SYSTEM ModbusExmpl
  (* Version 1.0, 2026-07-14, alex *)
  APPLICATION testttApp
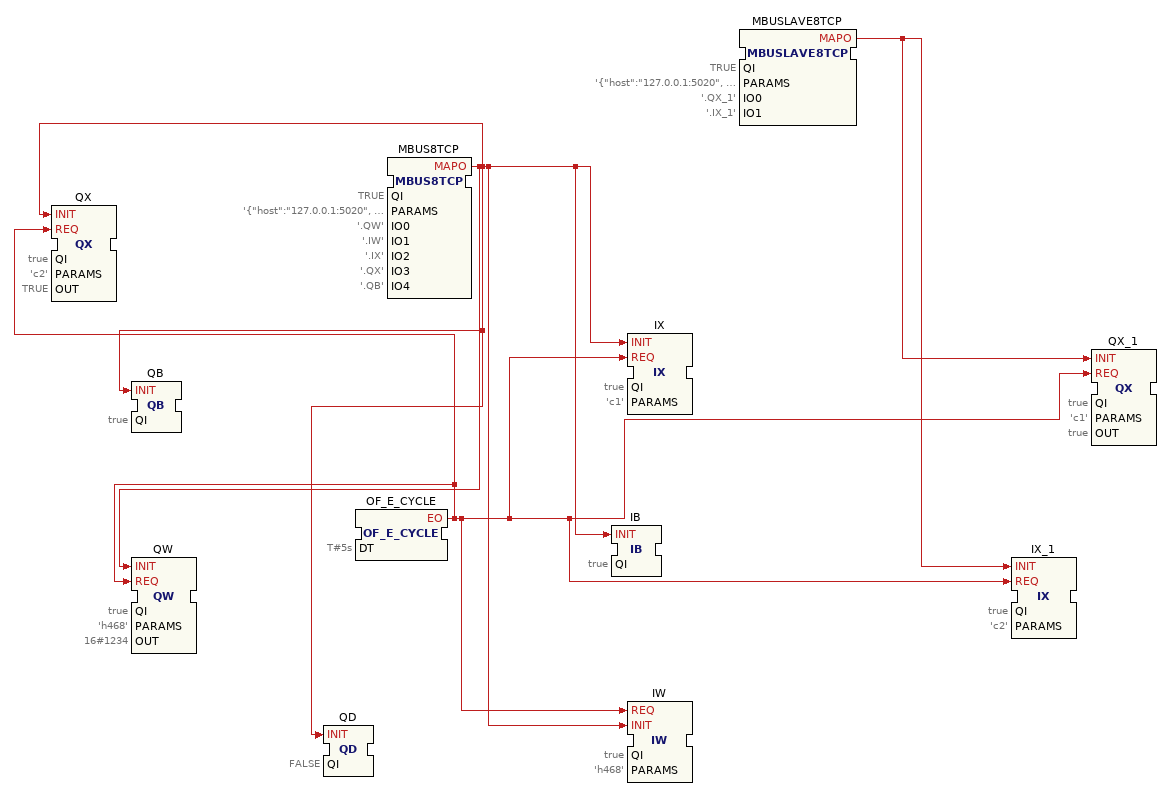
    FBS
      MBUS8TCP : MBUS8TCP(QI := TRUE, PARAMS := '{"host":"127.0.0.1:5020", "id":"1"}', IO0 := '.QW', IO1 := '.IW', IO2 := '.IX', IO3 := '.QX', IO4 := '.QB');
      MBUSLAVE8TCP : MBUSLAVE8TCP(QI := TRUE, PARAMS := '{"host":"127.0.0.1:5020", "id":"1"}', IO0 := '.QX_1', IO1 := '.IX_1');
      QX : QX(QI := true, PARAMS := 'c2', OUT := TRUE);
      QB : QB(QI := true);
      QD : QD(QI := FALSE);
      QW : QW(QI := true, PARAMS := 'h468', OUT := 16#1234);
      IX : IX(QI := true, PARAMS := 'c1');
      IB : IB(QI := true);
      IX_1 : IX(QI := true, PARAMS := 'c2');
      QX_1 : QX(QI := true, PARAMS := 'c1', OUT := true);
      OF_E_CYCLE : OF_E_CYCLE(DT := T#5s);
      IW : IW(QI := true, PARAMS := 'h468');
    END_FBS
    EVENT_CONNECTIONS
      MBUS8TCP.MAPO TO QX.INIT;
      MBUS8TCP.MAPO TO QB.INIT;
      MBUS8TCP.MAPO TO QW.INIT;
      MBUS8TCP.MAPO TO QD.INIT;
      MBUSLAVE8TCP.MAPO TO QX_1.INIT;
      MBUSLAVE8TCP.MAPO TO IX_1.INIT;
      MBUS8TCP.MAPO TO IX.INIT;
      MBUS8TCP.MAPO TO IB.INIT;
      OF_E_CYCLE.EO TO QX.REQ;
      OF_E_CYCLE.EO TO QW.REQ;
      OF_E_CYCLE.EO TO IX_1.REQ;
      OF_E_CYCLE.EO TO QX_1.REQ;
      OF_E_CYCLE.EO TO IX.REQ;
      OF_E_CYCLE.EO TO IW.REQ;
      MBUS8TCP.MAPO TO IW.INIT;
    END_CONNECTIONS
  END_APPLICATION
  DEVICE FORTE_PC : FORTE_PC(MGR_ID := "localhost:61499" (* Device manager socket ID *))
    {SET_ATTRIBUTE(Profile, HOLOBLOC)}
    RESOURCE EMB_RES : EMB_RES
    END_RESOURCE
  END_DEVICE
  MAPPINGS
    testttApp.MBUS8TCP ON FORTE_PC.EMB_RES;
    testttApp.MBUSLAVE8TCP ON FORTE_PC.EMB_RES;
    testttApp.IX_1 ON FORTE_PC.EMB_RES;
    testttApp.IX ON FORTE_PC.EMB_RES;
    testttApp.IB ON FORTE_PC.EMB_RES;
    testttApp.QX_1 ON FORTE_PC.EMB_RES;
    testttApp.QX ON FORTE_PC.EMB_RES;
    testttApp.QB ON FORTE_PC.EMB_RES;
    testttApp.QW ON FORTE_PC.EMB_RES;
    testttApp.QD ON FORTE_PC.EMB_RES;
    testttApp.OF_E_CYCLE ON FORTE_PC.EMB_RES;
    testttApp.IW ON FORTE_PC.EMB_RES;
  END_MAPPINGS
  SEGMENTS
    Ethernet : Ethernet;
  END_SEGMENTS
  LINKS
    FORTE_PC => Ethernet;
  END_LINKS
END_SYSTEM
